// TIA Portal V21 export
TYPE "OBJ_Timer_Type"
   STRUCT
      ixIN : Bool;
      ixRES : Bool;
      oxQ : Bool;
      ifPT : Real;
      ifValue : Real;
      "@Data" { ExternalAccessible := 'False'; ExternalVisible := 'False'; ExternalWritable := 'False'} : Struct
         xMem : Bool;
         xFP : Bool;
         fPT : Real;
         fAcc : Real;
      END_STRUCT;
   END_STRUCT;
END_TYPE
